// TIA Portal V17 export
// export: Created 2024-09-02T12:50:25.4472384Z, ExportSetting WithDefaults, DisplayName Totally Integrated Automation Portal, DisplayVersion V17, DisplayName TIA Portal Openness, DisplayVersion V17, DisplayName TIA Portal Version Control Interface, DisplayVersion V17, DisplayName STEP 7 Professional, DisplayVersion V17, DisplayName STEP 7 Safety, DisplayVersion V17, DisplayName WinCC Professional, DisplayVersion V17
VAR_GLOBAL   // PLC tag table "FeederUnit"
   I_M210_Loading_cylinder_Dumper_Cap_in_Up_pos AT %I55.0 : Bool;
   I_M210_Loading_cylinder_Dumper_Cap_in_Down_pos AT %I55.1 : Bool;
   i_Dumper_Cap_Part_in_Separator AT %I55.2 : Bool;
   i_Dumper_Cap_Part_in_Separator_Buffor AT %I55.3 : Bool;
   i_Dumper_Cap_Corect_Level_Of_Part AT %I55.4 : Bool;
   i_Dumper_Cap_Part_in_the_pipe AT %I55.5 : Bool;
   I_M220_Separation_cylinder_Dumper_Cap_in_Front_pos AT %I55.6 : Bool;
   I_M220_Separation_cylinder_Dumper_Cap_in_Back_pos AT %I55.7 : Bool;
   Q_M230_Air_for_blown_ON AT %Q51.0 : Bool;
   Q_M220_Separation_cylinder_Dumper_Cap_Forward AT %Q51.1 : Bool;
   Q_M220_Separation_cylinder_Dumper_Cap_Backward AT %Q51.5 : Bool;
   Q_M210_Loading_cylinder_Dumper_Cap_Upward AT %Q51.2 : Bool;
   Q_M210_Loading_cylinder_Dumper_Cap_Downward AT %Q51.6 : Bool;
   i_Screw_Corect_Level_Of_Part AT %I56.1 : Bool;
   i_Ball_Corect_Level_Of_Part AT %I56.0 : Bool;
   Q_Feeder_unit_Ball_Start AT %Q2.5 : Bool;
   Q_Feeder_unit_Screw_Start AT %Q2.6 : Bool;
   I_Feeder_unit_Screw_Alarm AT %I1.7 : Bool;
   I_Feeder_unit_Screw_Impuls AT %I1.6 : Bool;
   I_Feeder_unit_Ball_Alarm AT %I1.5 : Bool;
   I_Feeder_unit_Ball_Impuls AT %I1.4 : Bool;
   Q_Feeder_unit_ON AT %Q0.6 : Bool;   // Meldeleuchte Halt bei Taktende (+ZP01-600PF0.6)
   Q_Feeder_unit_Damper_Cap_Start AT %M500.0 : Bool;
   I_Screw_present_OP70 AT %I56.2 : Bool;
   Q_Feeder_Unit_Damper_Cap_ON AT %Q0.7 : Bool;
END_VAR
